(*********************************** G.D S.p.A. - Technical Department ***********************************
============= PROGRAM INFO ============
FOLDER:             TBD
MACHINES INVOLVED:  TBD 

============= DESCRIPTION =============
Low task

============= REVISIONS ===============
Date		Version	 	Author      	Description             
----------	-------		------------  	--------------------------------------------
2019/03/28 	0000.00	 	CEC 		Creation of the PRG

**********************************************************************************************************)

PROGRAM _csp_customerInterfaces_lowest
VAR
END_VAR

		csp_customerInterfaces();

END_PROGRAM

(* stored: Version 1.1.0.1, ProductVersion 3.1.4024.3
   POU _csp_customerInterfaces_lowest: Id {99ae9e08-2b3f-4579-85ba-7dcaf0bd855a}, SpecialFunc None *)
